{attribute addProperty BoxType "EP7402-0057-0017"}
{attribute addProperty Id "DI_InputsAT %I*DI_Inputs_3959EB256480STM_Status_Channel_1AT %I*STM_Status_Channel_48EC80151620STM_Synchron_info_data_Channel_1AT %I*STM_Synchron_info_data_Channel_A9A5537A4860STM_Status_Channel_2AT %I*STM_Status_Channel_48EC80151620STM_Synchron_info_data_Channel_2AT %I*STM_Synchron_info_data_Channel_A9A5537A4860STM_Inputs_DeviceAT %I*STM_Inputs_Device_9A6149C03240DO_OutputsAT %Q*DO_Outputs_43F80E286480STM_Control_Channel_1AT %Q*STM_Control_Channel_D4E6554C1620STM_Target_Velocity_Channel_1AT %Q*STM_Target_Velocity_Channel_40EDC30B4860STM_Control_Channel_2AT %Q*STM_Control_Channel_D4E6554C1620STM_Target_Velocity_Channel_2AT %Q*STM_Target_Velocity_Channel_40EDC30B4860WcStateAT %I*WcState_F855686C1620InfoDataAT %I*InfoData_3F3BB279112140"}
{attribute addProperty CRC "2651089185"}
{attribute addProperty SizeInBites "544"}
{attribute addProperty SizeInBytes "68"}
TYPE EP7402_B02F38FD :
STRUCT
	{attribute addProperty Name "DI_Inputs"}
	DI_Inputs : DI_Inputs_3959EB25;
	{attribute addProperty Name "STM_Status_Channel_1"}
	STM_Status_Channel_1 : STM_Status_Channel_48EC8015;
	{attribute addProperty Name "STM_Synchron_info_data_Channel_1"}
	STM_Synchron_info_data_Channel_1 : STM_Synchron_info_data_Channel_A9A5537A;
	{attribute addProperty Name "STM_Status_Channel_2"}
	STM_Status_Channel_2 : STM_Status_Channel_48EC8015;
	{attribute addProperty Name "STM_Synchron_info_data_Channel_2"}
	STM_Synchron_info_data_Channel_2 : STM_Synchron_info_data_Channel_A9A5537A;
	{attribute addProperty Name "STM_Inputs_Device"}
	STM_Inputs_Device : STM_Inputs_Device_9A6149C0;
	{attribute addProperty Name "DO_Outputs"}
	DO_Outputs : DO_Outputs_43F80E28;
	{attribute addProperty Name "STM_Control_Channel_1"}
	STM_Control_Channel_1 : STM_Control_Channel_D4E6554C;
	{attribute addProperty Name "STM_Target_Velocity_Channel_1"}
	STM_Target_Velocity_Channel_1 : STM_Target_Velocity_Channel_40EDC30B;
	{attribute addProperty Name "STM_Control_Channel_2"}
	STM_Control_Channel_2 : STM_Control_Channel_D4E6554C;
	{attribute addProperty Name "STM_Target_Velocity_Channel_2"}
	STM_Target_Velocity_Channel_2 : STM_Target_Velocity_Channel_40EDC30B;
	{attribute addProperty Name "WcState"}
	WcState : WcState_F855686C;
	{attribute addProperty Name "InfoData"}
	InfoData : InfoData_3F3BB279;
END_STRUCT
END_TYPE

(* stored: Version 1.2.0.0, ProductVersion 3.1.4024.9
   DUT EP7402_B02F38FD: Id {6f530533-a5e3-4012-ba44-9fdb2e8e7e53} *)
